// TIA Portal V20 export
// export: Created 2025-12-01T14:56:12.2670438Z, ExportSetting None, DisplayName Totally Integrated Automation Portal, DisplayVersion V20 Update 3, DisplayName TIA Portal Openness, DisplayVersion V20 Update 3, DisplayName TIA Portal Version Control Interface, DisplayVersion V20 Update 3, DisplayName STEP 7 Professional, DisplayVersion V20 Update 3, DisplayName STEP 7 Safety, DisplayVersion V20 Update 2, DisplayName WinCC Basic/Comfort/Advanced, DisplayVersion V20 Update 3, DisplayName WinCC Professional, DisplayVersion V20 Update 3, DisplayName WinCC Unified, DisplayVersion V20 Update 3
TYPE "UDT_ConfigFB"
   STRUCT
      Galibo : Bool := TRUE;   // Galibo Actual >> Año 2023
      Inicio_E1E3 : Bool := TRUE;   // Es Inicio de Transportador E1E3 >> E1 es Inicio
      Final_E1E3 : Bool := TRUE;   // Es Final de Transportador E1E3 >> E3 es Final
      Inicio_E2E4 : Bool := TRUE;   // Es Inicio de Transportador E2E4 >> E2 es Inicio
      Final_E2E4 : Bool := TRUE;   // Es Final de Transportador E2E4 >> E4 es Final
      Simultaneo_E1 : Bool;   // Permiso de Simultaneo en la Entrada E1
      Simultaneo_E2 : Bool;   // Permiso de Simultaneo en la Entrada E2
      Simultaneo_E3 : Bool;   // Permiso de Simultaneo en la Entrada E3
      Simultaneo_E4 : Bool;   // Permiso de Simultaneo en la Entrada E4
      NoEntrar_E0 : Bool;   // No Entrar Carga por E0
      NoEntrar_E1 : Bool;   // No Entrar Carga por E1
      NoEntrar_E2 : Bool;   // No Entrar Carga por E2
      NoEntrar_E3 : Bool;   // No Entrar Carga por E3
      NoEntrar_E4 : Bool;   // No Entrar Carga por E4
      Ausencia_S1 : Bool;   // Se enviara Ausencia cuando la carga sale por S1
      Ausencia_S2 : Bool;   // Se enviara Ausencia cuando la carga sale por S2
      Ausencia_S3 : Bool;   // Se enviara Ausencia cuando la carga sale por S3
      Ausencia_S4 : Bool;   // Se enviara Ausencia cuando la carga sale por S4
      SinErrorLiberarPHS_S1 : Bool;
      SinErrorLiberarPHS_S2 : Bool;
      SinErrorLiberarPHS_S3 : Bool;
      SinErrorLiberarPHS_S4 : Bool;
   END_STRUCT;
END_TYPE
